Staubli VAL3: page_viewInstr.pjx

--- page_viewInstr.pjx ---
Parameters version=s7.2.1 stackSize=5000 millimeterUnit=true
Program file=buildList.pgx
Program file=getItem.pgx
Program file=listAdd.pgx
Program file=loadPage.pgx
Program file=main.pgx
Program file=onEnterEvent.pgx
Program file=onExit.pgx
Program file=onF1Event.pgx
Program file=onF2Event.pgx
Program file=onF3Event.pgx
Program file=onF4Event.pgx
Program file=onF5Event.pgx
Program file=onF6Event.pgx
Program file=onF7Event.pgx
Program file=onF8Event.pgx
Program file=onStart.pgx
Program file=refresh.pgx
Program file=refreshDynamic.pgx
Program file=refreshStatic.pgx
Data file=page_viewInstr.dtx
Library alias=page path=Disk://kernel/template/page/page.pjx
Library alias=use path=Disk://kernel/userPage/userPage.pjx
Library alias=language path=Disk://kernel/language/language.pjx
Library alias=saveData path=Disk://saveData/saveData.pjx
Library alias=events path=Disk://..//templates/instruction/instruction.pjx
Library alias=prog path=Disk://instruction/PROG/PROG.pjx
Library alias=cycleStatus path=Disk://cycleStatus/cycleStatus.pjx
Library alias=TrajItem path=Disk://../templates/trajectory/trajectory.pjx
Library alias=sub path=Disk://instruction/SUB/SUB.pjx
Library alias=saveInputOutput path=Disk://saveInputOutput/saveInputOutput.pjx
Type name=InstrItem path=Disk://kernel/template/InstrItem/InstrItem.pjx
Type name=TrajectoryItem path=Disk://kernel/template/TrajectoryItem/TrajectoryItem.pjx
Type name=progItem path=Disk://kernel/template/progItem/progItem.pjx
Type name=dioItem path=Disk://kernel/template/dioItem/dioItem.pjx

--- page_viewInstr.dtx ---
num nIndex
num nKey
public num nPage
num nRefresh
num nSelected
num nTime = 1
num nView
string sEvent
public string sItems
string sList
string sMenu[8]
string sMessage
string sProgram
string sMenu8[8]
bool bButton[8]
  [0] = true
  [2] = true
  [3] = true
  [4] = true
  [5] = true
  [6] = true
  [7] = true
bool bLarge

--- main.pgx ---
public program main()
begin
  // INIT
  call onStart()
  //
  // LOOP UNTIL nKey=255
  do
    call refresh()
    nKey=getKey()
    call use:listevent(nKey,nIndex,sEvent)
    nView=use:nView
    nSelected=nIndex
    switch nKey
      case 259
        // TAB-> ENLARGE
        bLarge=!bLarge
        call use:setView(bLarge)
      break
      case 271
        // Simulation
        call onF1Event()
      break
      case 272
        call onF2Event()
      break
      case 273
        call onF3Event()
      break
      case 274
        call onF4Event()
      break
      case 275
        call onF5Event()
      break
      case 276
        call onF6Event()
      break
      case 277
        call onF7Event()
      break
      case 278
        call onF8Event()
      break
      case 270
        call onEnterEvent()
      break
    endSwitch
    //release the resource
    delay(0)
  until nKey==255
  // on Exit
  call onExit()
end

--- getItem.pgx ---
program getItem(string& x_sItem[], num x_nIndex)
begin
  x_sItem=sList[x_nIndex]
end

--- onEnterEvent.pgx ---
program onEnterEvent()
begin
  //
end

--- onExit.pgx ---
program onExit()
  local string l_sMessage
begin
  //
end

--- onF1Event.pgx ---
program onF1Event()
  local bool l_bYes
  local string l_sMessage
  local InstrItem l_iItem
  local string l_sButton[2]
  local string l_sPage
begin
  // look if the bButton is enable
  if bButton[0]
    //
    //
    // the SIMULATION is disable when cycle is active
    //
    if !cycleStatus:bCycle
      call language:message(l_sMessage,214)
      // get the yes_no button Key
      call language:getYesNo(l_sButton)
      // ask the question
      call use:yes_no(l_sMessage,l_sButton,l_bYes)
      if l_bYes
        call prog:getItem(l_iItem,nIndex)
        cycleStatus:iToSuperV=l_iItem
        cycleStatus:nInterfaceToSV=3
        logMsg("[KERNEL] INTERFACE:Simulation of the item: "+sEvent)
        wait(cycleStatus:nInterfaceToSV==-1)
        // load the production page
        l_sPage="simulation"
        call loadPage("kernel/page/production",l_sPage)
        call use:setView(false)
      endIf
    endIf
  endIf
end

--- onF2Event.pgx ---
program onF2Event()
  local string l_sMessage
  local bool l_bYes
  local num i
begin
  // look if the bButton is enable
  if bButton[1]
    //
  endIf
end

--- onF3Event.pgx ---
program onF3Event()
  local string l_sMessage
  local bool l_bYes
  local num i
begin
  // look if the bButton is enable
  if bButton[2]
    //
  endIf
end

--- onF4Event.pgx ---
program onF4Event()
begin
  // look if the bButton is enable
  if bButton[3]
    //
  endIf
end

--- onF5Event.pgx ---
program onF5Event()
begin
  // look if the bButton is enable
  if bButton[4]
    //
  endIf
end

--- onF6Event.pgx ---
program onF6Event()
  local bool l_bYes
  local string l_sMessage
begin
  // look if the bButton is enable
  if bButton[5]
    //
  endIf
end

--- onF7Event.pgx ---
program onF7Event()
  local num l_nIndex
  local string l_sItem
  local num i
  local num l_nResult
  local string l_sMessage
begin
  // look if the bButton is enable
  if bButton[6]
    //
  endIf
end

--- onF8Event.pgx ---
program onF8Event()
  local num x_nResult
begin
  // look if the bButton is enable
  if bButton[7]
    //
  endIf
end

--- onStart.pgx ---
program onStart()
  local num i
  local string l_sMessage
begin
  // reset the index
  nIndex=nSelected=nView=0
  // reset the Key pressure
  call use:nullKey(nKey)
  // logMsg
  logMsg("[KERNEL] INTERFACE:PAGE view program")
  //
  sProgram=sItems[0]
  //
  call prog:load(sProgram,i)
  if i!=0
// error loading
    call language:message(l_sMessage,-7)
    popUpMsg(l_sMessage+" PROG "+sProgram+" code "+toString("",i))
  endIf
  // define the list
  call buildList()
  // build the page
  call refreshStatic()
  logMsg("ON MEMORY events INSTRUCTION "+events:libPath())
end

--- refreshStatic.pgx ---
program refreshStatic()
  local string l_sMessage
  local string l_sEvent
  local num i
  local num l_nSize
begin
  cls()
  //
  // set the view of the page..
  //
  // SET THE PAGE NUMBER
  use:nPage=10010
  // USE <>PROFILE for <>PAGE
  use:nPage=use:nPage+abs(limit(saveData:mode,0,2)-2)
  if cycleStatus:bCycle
    use:nPage=use:nPage+3
  endIf
  // load the menu page
  if saveData:language!="japanese"
    // SET THE VIEW OF THE PAGE
    call language:page(l_sMessage,use:nPage)
    // define the menu
    call use:stringToArray(l_sMessage,sMenu)
    call use:setMenu(sMenu,true,3)
  else
    // japanese use the array for the menu
    call language:page(sMenu8,use:nPage)
    call use:stringCopy(sMenu8,sMenu)
    call use:setMenu(sMenu,false,3)
  endIf
  //
  if sProgram==""
    // save or not
    sMenu[7]=""
  endIf
  // set the menu
  if saveData:language!="japanese"
    call use:setMenu(sMenu,true,3)
  else
    call use:setMenu(sMenu,false,3)
  endIf
  call use:getMenu(sMenu,bButton)
  //
  // CREATE THE LIST
  //
  // define your list size for default
  call use:setSizeList(19,0,19,11)
  call use:setView(bLarge)
  //
  call use:listcreate("PROG "+sProgram)
  //
  call prog:getSizeItem(l_nSize)
  for i=0 to l_nSize-1
    l_sEvent=sList[i]
    call use:listadd(l_sEvent)
  endFor
  //
  // refresh
  call use:selectNewField(nSelected,nIndex,nView)
  nSelected=-1
end
